{attribute 'to_string'}
TYPE E_ErrorHandling :
(
	Fault := 900,
	Emergency := 999,
	No_Error := 0
);
END_TYPE

(* stored: Version 1.1.0.1
   DUT E_ErrorHandling: Id {3d2743bc-551a-4847-9164-fffcd0546ff1} *)
